(********************* G.D S.p.A. - Technical Department ***********************************
This program has been generated automatically from Application Designer DE&F
********************************************************************************************)
PROGRAM dbg_csp_case_fc_os_upper_follower
VAR
  axis_shd : axis_shadow;
END_VAR

_objects_manager();

IF	g_application_status <> APPLICATION_STATUS_RUNNING
THEN
	RETURN;
END_IF

CASE process_get_mode(CONVERSION_this := dbg_root.prc) OF
	MODE_ABSENT,
	MODE_INACTIVE:
		RETURN;
	MODE_TEST:
		RETURN;
END_CASE

ACTION _objects_manager:
IF	objects_initialization()
THEN
	axis_shadow_init(
		sim_mode:= SHADOW_SIMULATION_MODE_AUTOMATIC, 
		father:= csp_case_fc_os_upper_follower.axis, 
		process:= dbg_root.prc, 
		CONVERSION_this:= axis_shd);

	RETURN;
END_IF

IF	objects_running()
THEN
	axis_shadow_cycle(axis_shd);
END_IF
END_ACTION

END_PROGRAM

(* stored: Version 1.1.0.1, ProductVersion 3.1.4022.12
   POU dbg_csp_case_fc_os_upper_follower: Id {35f98b1f-1c7f-4402-bf76-46161cb45d18}, SpecialFunc None
   Action _objects_manager: Id {2c39d83d-4881-47ad-b1cc-0c39424595bd} *)
